TYPE ST_SettingsDoorLock :
STRUCT
	tReleasingLockTimeout : TIME := T#30S;	/// Timeout for releasing lock [default: 3s]
	tApplyingLockTimeout : TIME := T#30S;	/// Timeout for applying door [default: 3s]
END_STRUCT
END_TYPE

(* stored: Version 1.1.0.1, ProductVersion 3.1.4024.12
   DUT ST_SettingsDoorLock: Id {959adbfb-3b17-44ae-9aa1-564241597ba9} *)
